// Mitsubishi GX Works2 project: GX W2 L6 Ex 2 DK C   PLC: FX3G

// global labels: Global1
VAR_GLOBAL
  oBorder AT Y000 : BOOL;
  iStart_PB AT X002 : BOOL;
  oO_Letter AT Y001 : BOOL;
  oP_Letter AT Y002 : BOOL;
  oE_Letter AT Y003 : BOOL;
  oN_Letter AT Y004 : BOOL;
END_VAR

// task Task_01 (event TRUE, interval 0, priority 31): POU_01

PROGRAM POU_01
VAR
  wSequence_States : INT;
  TON_1 : TON;
  TON_2 : TON;
  TON_3 : TON;
  TON_4 : TON;
  TON_5 : TON;
END_VAR
(* structured ladder/FBD written out as ST: instructions are called as NAME(EN, inputs, outputs); _pN, _eN, _tN stand for wires *)
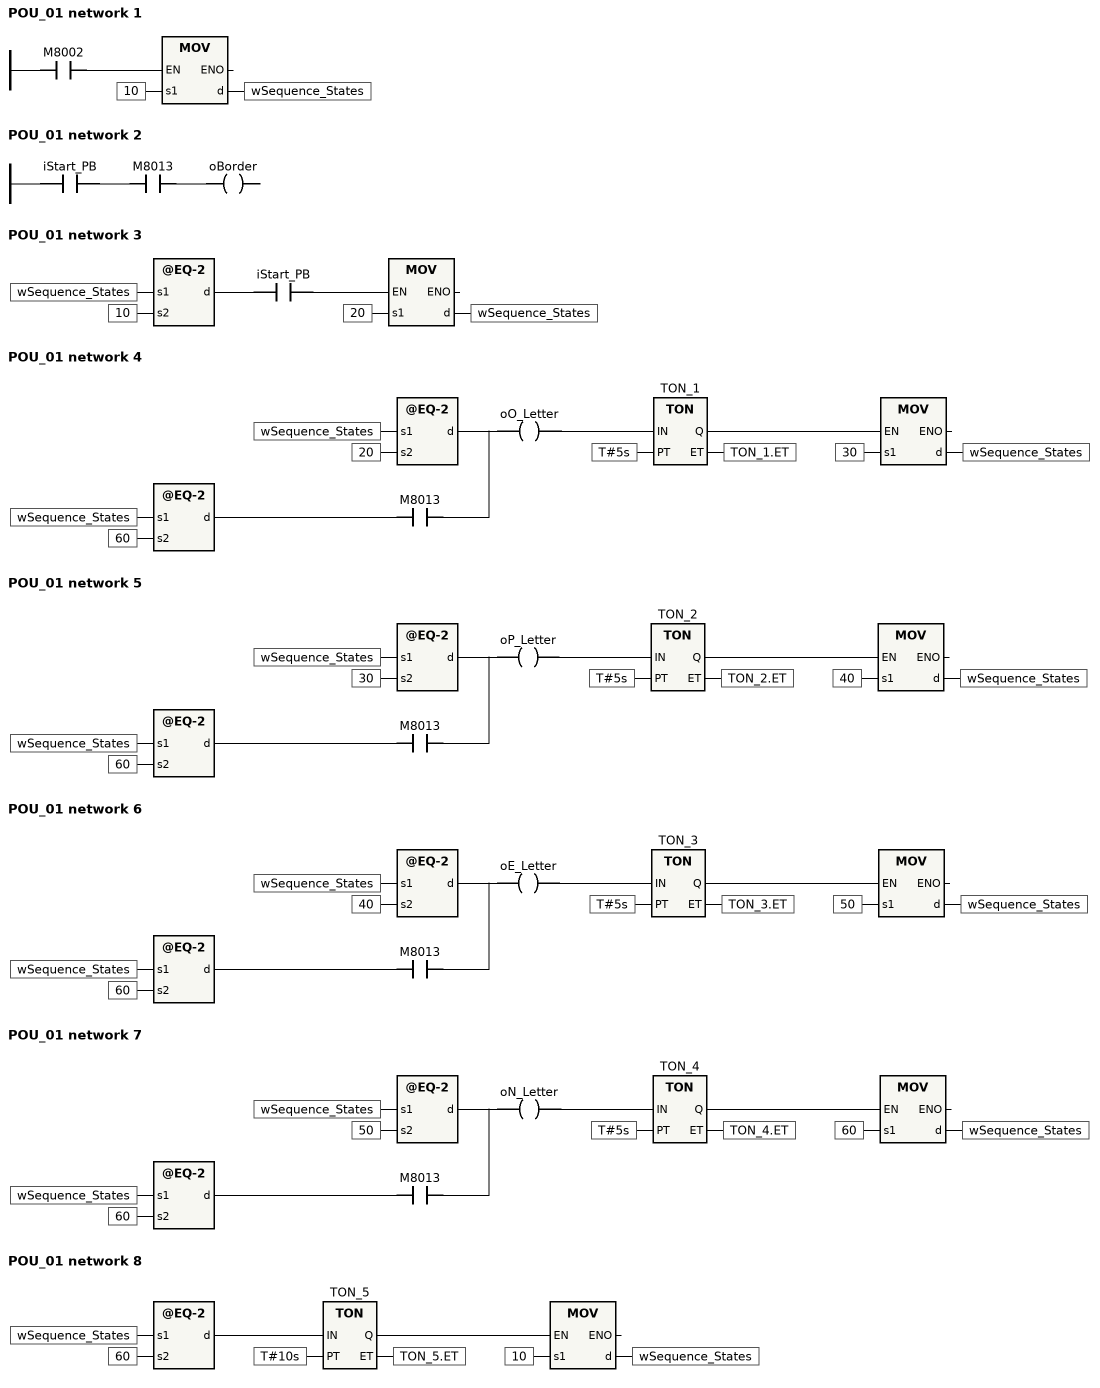
(* network 1 *)
MOV(M8002, 10, wSequence_States);
(* network 2 *)
oBorder := iStart_PB AND M8013;
(* network 3 *)
MOV(@EQ-2(wSequence_States, 10) AND iStart_PB, 20, wSequence_States);
(* network 4 *)
_p1 := (@EQ-2(wSequence_States, 20)) OR (@EQ-2(wSequence_States, 60) AND M8013);
oO_Letter := _p1;
TON_1(IN := _p1, PT := T#5s, ET => TON_1.ET);
MOV(TON_1.Q, 30, wSequence_States);
(* network 5 *)
_p1 := (@EQ-2(wSequence_States, 30)) OR (@EQ-2(wSequence_States, 60) AND M8013);
oP_Letter := _p1;
TON_2(IN := _p1, PT := T#5s, ET => TON_2.ET);
MOV(TON_2.Q, 40, wSequence_States);
(* network 6 *)
_p1 := (@EQ-2(wSequence_States, 40)) OR (@EQ-2(wSequence_States, 60) AND M8013);
oE_Letter := _p1;
TON_3(IN := _p1, PT := T#5s, ET => TON_3.ET);
MOV(TON_3.Q, 50, wSequence_States);
(* network 7 *)
_p1 := (@EQ-2(wSequence_States, 50)) OR (@EQ-2(wSequence_States, 60) AND M8013);
oN_Letter := _p1;
TON_4(IN := _p1, PT := T#5s, ET => TON_4.ET);
MOV(TON_4.Q, 60, wSequence_States);
(* network 8 *)
TON_5(IN := @EQ-2(wSequence_States, 60), PT := T#10s, ET => TON_5.ET);
MOV(TON_5.Q, 10, wSequence_States);
END_PROGRAM
